// TIA Portal V20 export
// export: Created 2025-12-01T14:57:46.1717008Z, ExportSetting None, DisplayName Totally Integrated Automation Portal, DisplayVersion V20 Update 3, DisplayName TIA Portal Openness, DisplayVersion V20 Update 3, DisplayName TIA Portal Version Control Interface, DisplayVersion V20 Update 3, DisplayName STEP 7 Professional, DisplayVersion V20 Update 3, DisplayName STEP 7 Safety, DisplayVersion V20 Update 2, DisplayName WinCC Basic/Comfort/Advanced, DisplayVersion V20 Update 3, DisplayName WinCC Professional, DisplayVersion V20 Update 3, DisplayName WinCC Unified, DisplayVersion V20 Update 3
DATA_BLOCK "DB201_RegEtiquetas_0001_1000"   // DB201
{ S7_Optimized_Access := 'FALSE' }
AUTHOR : ROUTER
NAME : 20130623
VERSION : 3.1
// stored: AutoNumber false
   VAR
      Reg_Etiqueta { S7_SetPoint := 'True'} : Array[1.."ROUT_Cantidad_Etiquetas_DB"] of "ROUT_Reg_Etiqueta";
   END_VAR
BEGIN
END_DATA_BLOCK
